PROGRAM prFeedScrewS5
VAR
    SolFeed : fbSingleSolRy;
    ErrorState : BOOL;
    AutoFlow : INT;
    TON1 : TON;
    TON2 : TON;
    TON3 : TON;
    Check1 : fbCheckScrew_Tube;
    Check2 : fbCheckScrew_Tube;
    RTRIG1 : R_TRIG;
END_VAR
VAR_EXTERNAL
    AutoStatus : bool;
    SystemReadyStatus : bool;
    HMIPB_SOL_S5_Feed : BOOL;
    SOL_S5_Feed : BOOL;
    FeedStartFlag : ARRAY[0..1] OF bool;
    HMI_FeedScrewTime : ARRAY[0..1] OF INT;
    RY_S5_Feed : BOOL;
    OutPutFeedRYS5 : BOOL;
    LS_S5_UpDownOut : BOOL;
    SNR_S5_L_Feed : BOOL;
    PB_Reset1 : BOOL;
    PB_Reset2 : BOOL;
    Error_SNR_S5_L_Feed : BOOL;
    SNR_S5_R_Feed : BOOL;
    Error_SNR_S5_R_Feed : BOOL;
    OBJScrewInClip : ARRAY[0..3] OF INT;
    OBJScrewInTube : ARRAY[0..3] OF INT;
    LS_S5_UpDownBack : BOOL;
    SOL_S5_UpDown : BOOL;
    HMIPB_S5Feed : BOOL;
END_VAR
//********************************************************************
//Check
//********************************************************************
Check1(
	inClearSingle:=LS_S5_UpDownOut,
	inFeedSNR:=SNR_S5_L_Feed,
	inBlowSOL:=SOL_S5_Feed,
	inReset:=PB_Reset1 OR PB_Reset2,
	outError=>Error_SNR_S5_L_Feed,
	inoutScrewInClip:=OBJScrewInClip[0],
	inoutScrewInTube:=OBJScrewInTube[0]);
Check2(
	inClearSingle:=LS_S5_UpDownOut,
	inFeedSNR:=SNR_S5_R_Feed,
	inBlowSOL:=SOL_S5_Feed,
	inReset:=PB_Reset1 OR PB_Reset2,
	outError=>Error_SNR_S5_R_Feed,
	inoutScrewInClip:=OBJScrewInClip[1],
	inoutScrewInTube:=OBJScrewInTube[1]);
//********************************************************************
//Manual
//********************************************************************
//Feed screw sol
SolFeed(
	inAutoStatus:=AutoStatus,
	inAutoFlowSet:=AutoFlow=3,
	inAutoFlowReset:=AutoFlow=4,
	inInterLockBack:=TRUE,
	inInterLockOut:=NOT(SOL_S5_UpDown) AND LS_S5_UpDownBack,
	outSol=>	SOL_S5_Feed);
//********************************************************************
//Auto
//********************************************************************
IF LS_S5_UpDownOut AND SOL_S5_UpDown THEN
	FeedStartFlag[0]:=TRUE;
END_IF;
ErrorState:=FALSE;
//power on=0
IF NOT(SystemReadyStatus) OR ErrorState THEN
	AutoFlow:=0;
	FeedStartFlag[0]:=FALSE;
END_IF;
//idle=1
IF AutoFlow=0 AND NOT(NOT(SystemReadyStatus) OR ErrorState) THEN
	AutoFlow:=1;
END_IF;
IF AutoFlow=6 AND NOT(OutPutFeedRYS5) THEN
	AutoFlow:=1;
END_IF;
//Feed RY on=2
RTRIG1(Clk:=HMIPB_SOL_S5_Feed);
IF AutoFlow=1 AND ((FeedStartFlag[0] AND AutoStatus) OR (RTRIG1.Q AND NOT(AutoStatus))) THEN
	AutoFlow:=2;
	OutPutFeedRYS5:=TRUE;
END_IF;
//Feed Sol on=3
TON1(In:=AutoFlow=2 AND RY_S5_Feed, PT:=t#800ms);
//
IF AutoFlow=2 AND TON1.Q THEN
	AutoFlow:=3;
END_IF;
IF AutoFlow=5 AND NOT(TON3.Q) AND FeedStartFlag[0] THEN
	AutoFlow:=3;
END_IF;
//Feed Sol off=4
TON2(In:=AutoFlow=3 AND SOL_S5_Feed, PT:=NanoSecToTime(HMI_FeedScrewTime[0]*100000000));
IF AutoFlow=3 AND ((TON2.Q AND AutoStatus) OR RTRIG1.Q AND NOT(AutoStatus)) THEN
	AutoFlow:=4;
END_IF;
//Feed Finish=5
IF AutoFlow=4 AND NOT(SOL_S5_Feed) THEN
	AutoFlow:=5;
	FeedStartFlag[0]:=FALSE;
END_IF;
//Feed RY off=6
TON3(In:=AutoFlow=5, PT:=t#5s);
IF AutoFlow=5 AND TON3.Q THEN
	AutoFlow:=6;
	OutPutFeedRYS5:=FALSE;
END_IF;
END_PROGRAM

PROGRAM prFeedScrewS6
VAR
    SolFeed : fbSingleSolRy;
    ErrorState : BOOL;
    AutoFlow : INT;
    TON1 : TON;
    TON2 : TON;
    TON3 : TON;
    Check1 : fbCheckScrew_Tube;
    Check2 : fbCheckScrew_Tube;
    RTRIG1 : R_TRIG;
END_VAR
VAR_EXTERNAL
    AutoStatus : bool;
    SystemReadyStatus : bool;
    HMIPB_SOL_S5_Feed : BOOL;
    SOL_S5_Feed : BOOL;
    FeedStartFlag : ARRAY[0..1] OF bool;
    HMI_FeedScrewTime : ARRAY[0..1] OF INT;
    RY_S5_Feed : BOOL;
    OutPutFeedRYS5 : BOOL;
    LS_S5_UpDownOut : BOOL;
    SNR_S5_L_Feed : BOOL;
    PB_Reset1 : BOOL;
    PB_Reset2 : BOOL;
    Error_SNR_S5_L_Feed : BOOL;
    SNR_S5_R_Feed : BOOL;
    Error_SNR_S5_R_Feed : BOOL;
    LS_S6_UpDownOut : BOOL;
    SNR_S6_L_Feed : BOOL;
    SOL_S6_Feed : BOOL;
    Error_SNR_S6_L_Feed : BOOL;
    SNR_S6_R_Feed : BOOL;
    Error_SNR_S6_R_Feed : BOOL;
    HMIPB_SOL_S6_Feed : BOOL;
    RY_S6_Feed : BOOL;
    OutPutFeedRYS6 : BOOL;
    OBJScrewInClip : ARRAY[0..3] OF INT;
    OBJScrewInTube : ARRAY[0..3] OF INT;
    LS_S6_UpDownBack : BOOL;
    SOL_S2_Fix : BOOL;
    SOL_S6_UpDown : BOOL;
END_VAR
//********************************************************************
//Check
//********************************************************************
Check1(
	inClearSingle:=LS_S6_UpDownOut,
	inFeedSNR:=SNR_S6_L_Feed,
	inBlowSOL:=SOL_S6_Feed,
	inReset:=PB_Reset1 OR PB_Reset2,
	outError=>Error_SNR_S6_L_Feed,
	inoutScrewInClip:=OBJScrewInClip[2],
	inoutScrewInTube:=OBJScrewInTube[2]);
Check2(
	inClearSingle:=LS_S6_UpDownOut,
	inFeedSNR:=SNR_S6_R_Feed,
	inBlowSOL:=SOL_S6_Feed,
	inReset:=PB_Reset1 OR PB_Reset2,
	outError=>Error_SNR_S6_R_Feed,
	inoutScrewInClip:=OBJScrewInClip[3],
	inoutScrewInTube:=OBJScrewInTube[3]);
//********************************************************************
//Manual
//********************************************************************
//Feed screw sol
SolFeed(
	inAutoStatus:=AutoStatus,
	inAutoFlowSet:=AutoFlow=3,
	inAutoFlowReset:=AutoFlow=4,
	inInterLockBack:=TRUE,
	inInterLockOut:=NOT(SOL_S6_UpDown) AND LS_S6_UpDownBack,
	outSol=>	SOL_S6_Feed);
//********************************************************************
//Auto
//********************************************************************
IF LS_S6_UpDownOut AND SOL_S6_UpDown THEN
	FeedStartFlag[1]:=TRUE;
END_IF;
ErrorState:=FALSE;
//power on=0
IF NOT(SystemReadyStatus) OR ErrorState THEN
	AutoFlow:=0;
	FeedStartFlag[1]:=FALSE;
END_IF;
//idle=1
IF AutoFlow=0 AND NOT(NOT(SystemReadyStatus) OR ErrorState) THEN
	AutoFlow:=1;
END_IF;
IF AutoFlow=6 AND NOT(OutPutFeedRYS6) THEN
	AutoFlow:=1;
END_IF;
//Feed RY on=2
RTRIG1(Clk:=HMIPB_SOL_S6_Feed);
IF AutoFlow=1 AND ((FeedStartFlag[1] AND AutoStatus) OR (RTRIG1.Q AND NOT(AutoStatus))) THEN
	AutoFlow:=2;
	OutPutFeedRYS6:=TRUE;
END_IF;
//Feed Sol on=3
TON1(In:=AutoFlow=2 AND RY_S6_Feed, PT:=t#800ms);
//
IF AutoFlow=2 AND TON1.Q THEN
	AutoFlow:=3;
END_IF;
IF AutoFlow=5 AND NOT(TON3.Q) AND FeedStartFlag[1] THEN
	AutoFlow:=3;
END_IF;
//Feed Sol off=4
TON2(In:=AutoFlow=3 AND SOL_S6_Feed, PT:=NanoSecToTime(HMI_FeedScrewTime[1]*100000000));
IF AutoFlow=3 AND ((TON2.Q AND AutoStatus) OR RTRIG1.Q AND NOT(AutoStatus)) THEN
	AutoFlow:=4;
END_IF;
//Feed Finish=5
IF AutoFlow=4 AND NOT(SOL_S6_Feed) THEN
	AutoFlow:=5;
	FeedStartFlag[1]:=FALSE;
END_IF;
//Feed RY off=6
TON3(In:=AutoFlow=5, PT:=t#5s);
IF AutoFlow=5 AND TON3.Q THEN
	AutoFlow:=6;
	OutPutFeedRYS6:=FALSE;
END_IF;
END_PROGRAM

PROGRAM prCommProgram
VAR
    statusFlash1s : BOOL;
    bClock : BOOL;
    TON1 : TON;
    TON2 : TON;
    R_TRIG1 : R_TRIG;
END_VAR
VAR_EXTERNAL
    Flash1s : BOOL;
    HMIPB_ResetCount : BOOL;
    HMI_AllCount : UDINT;
END_VAR
//bClock:=Get1sClk();
IF HMIPB_ResetCount THEN
	HMI_AllCount:=0;
END_IF;
//flsash 1s
TON1(In:=NOT(statusFlash1s), PT:=t#1s);
TON2(In:=(statusFlash1s), PT:=t#1s);
IF TON1.Q THEN
	bClock:=TRUE;
END_IF;
IF TON2.Q THEN
	bClock:=FALSE;
END_IF;
Flash1s:=bClock;
statusFlash1s:=Flash1s;
END_PROGRAM

PROGRAM prBZAndLight
VAR_EXTERNAL
    Flash1s : BOOL;
    GL : BOOL;
    YL : BOOL;
    SystemReadyStatus : bool;
    ErrorStatus_MachineNonStop : bool;
    ErrorStatus_MachineStop : bool;
    RL : BOOL;
    BZ : BOOL;
    MachineRunStatus : bool;
END_VAR
(*BZ*)	
IF (ErrorStatus_MachineStop OR ErrorStatus_MachineNonStop) THEN
	BZ:=Flash1s;
	ELSE
	BZ:=FALSE;
END_IF;
//(*紅燈長亮:異常*)
IF SystemReadyStatus AND (ErrorStatus_MachineStop) THEN
	RL:=TRUE;
	ELSE
	RL:=FALSE;
END_IF;
(*綠燈閃爍:運轉,長亮:待機*)
IF SystemReadyStatus AND NOT(ErrorStatus_MachineNonStop) AND NOT(ErrorStatus_MachineStop)  THEN
	IF MachineRunStatus THEN
		GL:=Flash1s;
	ELSE
		GL:=TRUE;
	END_IF;
	ELSE
	GL:=FALSE;
END_IF;
(*黃燈閃爍:振動筒缺料*)
IF SystemReadyStatus AND ErrorStatus_MachineNonStop AND NOT(ErrorStatus_MachineStop) THEN
	YL:=Flash1s;
	ELSE
	YL:=FALSE;
END_IF;
END_PROGRAM

PROGRAM prCycleTime
VAR
    TON1 : TON;
    tCycleTime : TIME;
    RTRIG1 : R_TRIG;
    cycle : LINT;
    FTRIG1 : F_TRIG;
END_VAR
VAR_EXTERNAL
    HMI_CycleTime : LINT;
    MachineRunStatus : bool;
    SNR_Index : BOOL;
END_VAR
IF FTRIG1.Q THEN
	HMI_CycleTime:=cycle;
END_IF;
TON1(In:=MachineRunStatus AND SNR_Index, PT:=t#1m,ET=>tCycleTime);
IF MachineRunStatus AND SNR_Index THEN
	cycle:=TimeToNanoSec(tCycleTime)/10000000;
END_IF;
FTRIG1(Clk:=SNR_Index);
END_PROGRAM

FUNCTION fIndexDataChange : BOOL
VAR_EXTERNAL
    IndexData8 : StationRecord;
    IndexData7 : StationRecord;
    IndexData6 : StationRecord;
    IndexData5 : StationRecord;
    IndexData4 : StationRecord;
    IndexData3 : StationRecord;
    IndexData2 : StationRecord;
    IndexData1 : StationRecord;
    IndexData0 : StationRecord;
END_VAR
IndexData8:=IndexData7;
IndexData7:=IndexData6;
IndexData6:=IndexData5;
IndexData5:=IndexData4;
IndexData4:=IndexData3;
IndexData3:=IndexData2;
IndexData2:=IndexData1;
IndexData1:=IndexData0;
END_FUNCTION

FUNCTION_BLOCK fbBowlFeeder
VAR
    AutoFlow : INT;
    TON_Auto1 : TON;
    TON_Auto2 : TON;
    TON_Auto3 : TON;
    tItemNotExistDelayTime : TIME;
    tItemExistTime : TIME;
    tItemNotExistErrorTime : TIME;
END_VAR
VAR_INPUT
    bFullSNR : BOOL;
    iItemNotExistDelayTime : LINT;
    iItemExistTime : LINT;
    iItemNotExistErrorTime : LINT;
END_VAR
VAR_OUTPUT
    bFullRY : BOOL;
    bFullSNRError : BOOL;
END_VAR
VAR_EXTERNAL
    SystemReadyStatus : BOOL;
END_VAR
(******************************************************************
程式:振動筒程序
作者:蔡相偉
版本資訊:v1.0		2016/4/16
******************************************************************)
//時間轉換
tItemNotExistDelayTime:=NanoSecToTime(In:=iItemNotExistDelayTime*100000000);
tItemExistTime:=NanoSecToTime(In:=iItemExistTime*100000000);
tItemNotExistErrorTime:=NanoSecToTime(In:=iItemNotExistErrorTime*100000000);
(*流程*)
(*PowerOn=0*)
IF NOT(SystemReadyStatus) THEN
	AutoFlow:=0;
END_IF;

(*Idle=1*)
IF AutoFlow=0 AND SystemReadyStatus THEN
	AutoFlow:=1;
END_IF;

IF AutoFlow=3 THEN
	AutoFlow:=1;
END_IF;

(*振動筒起振=2*)
TON_Auto1(IN:=AutoFlow=1 AND NOT(bFullSNR) , PT:=tItemNotExistDelayTime);
IF AutoFlow=1 AND TON_Auto1.Q THEN
	AutoFlow:=2;
END_IF;

(*振動筒停振=3*)
TON_Auto2(IN:=AutoFlow=2 AND bFullSNR , PT:=tItemExistTime);
TON_Auto3(IN:=NOT(bFullSNR) AND bFullRY, PT:=tItemNotExistErrorTime);
IF AutoFlow=2 AND TON_Auto2.Q THEN
	AutoFlow:=3;
END_IF;
(******************************************************************)
(*輸出*)
(*振動筒繼電器*)
IF AutoFlow=2 THEN
	bFullRY:=TRUE;
	ELSE
	bFullRY:=FALSE;
END_IF;
(*振動筒滿料異常*)
IF AutoFlow=2 AND (TON_Auto3.Q) THEN
	bFullSNRError:=TRUE;
	ELSE
	bFullSNRError:=FALSE;
END_IF;
END_FUNCTION_BLOCK

FUNCTION_BLOCK fbSingleSolRy
VAR
    solStatus : BOOL;
    R_TRIG1 : R_TRIG;
END_VAR
VAR_INPUT
    inPushButton : BOOL;
    inAutoStatus : BOOL;
    inAutoFlowSet : BOOL;
    inAutoFlowReset : BOOL;
    inInterLockBack : BOOL;
    inInterLockOut : BOOL;
END_VAR
VAR_OUTPUT
    outSol : BOOL;
END_VAR
(*電磁閥*)
R_TRIG1(Clk:=inPushButton AND NOT(inAutoStatus));
(*SET*)
IF ((R_TRIG1.Q AND NOT(solStatus)) OR inAutoFlowSet) AND inInterLockOut THEN
	outSol:=TRUE;
END_IF;
(*RESET*)
IF ((R_TRIG1.Q AND (solStatus)) OR inAutoFlowReset) AND inInterLockBack THEN
	outSol:=FALSE;
END_IF;
(*STATUS*)
solStatus:=outSol;
END_FUNCTION_BLOCK

FUNCTION_BLOCK fbErrorSOL_S
VAR
    TON_1 : TON;
    TON_2 : TON;
END_VAR
VAR_INPUT
    bAutoStatus : BOOL;
    bResetPB : BOOL;
    bSOL : BOOL;
    bBackLS : BOOL;
    bOutLS : BOOL;
END_VAR
VAR_OUTPUT
    bErrorStatus_Back : BOOL;
    bErrorStatus_Out : BOOL;
END_VAR
IF bAutoStatus AND NOT(bResetPB) THEN
	(*歸磁簧開關*)
	TON_1(IN:=(NOT(bSOL) AND NOT(bBackLS)) OR ((bSOL) AND bBackLS), PT:=t#2s);
	IF TON_1.Q THEN
		bErrorStatus_Back:=TRUE;
	END_IF;
	(*出磁簧開關*)
	TON_2(IN:=(NOT(bSOL) AND (bOutLS)) OR ((bSOL) AND NOT(bOutLS)), PT:=t#2s);
	IF TON_2.Q THEN
		bErrorStatus_Out:=TRUE;
	END_IF;
END_IF;
IF bResetPB THEN
	bErrorStatus_Back:=FALSE;
	bErrorStatus_Out:=FALSE;
END_IF;
END_FUNCTION_BLOCK

FUNCTION_BLOCK fbErrorSOL_D
VAR
    TON_1 : TON;
    TON_2 : TON;
END_VAR
VAR_INPUT
    bAutoStatus : BOOL;
    bResetPB : BOOL;
    bBackSOL : BOOL;
    bOutSOL : BOOL;
    bBackLS : BOOL;
    bOutLS : BOOL;
END_VAR
VAR_OUTPUT
    bErrorStatus_Back : BOOL;
    bErrorStatus_Out : BOOL;
END_VAR
IF bAutoStatus AND NOT(bResetPB) THEN
	(*歸磁簧開關*)
	TON_1(IN:=bBackSOL AND NOT(bBackLS), PT:=t#4s);
	IF TON_1.Q THEN
		bErrorStatus_Back:=TRUE;
	END_IF;
	(*出磁簧開關*)
	TON_2(IN:=bOutSOL AND NOT(bOutLS), PT:=t#4s);
	IF TON_2.Q THEN
		bErrorStatus_Out:=TRUE;
	END_IF;
END_IF;
IF bResetPB THEN
	bErrorStatus_Back:=FALSE;
	bErrorStatus_Out:=FALSE;
END_IF;
END_FUNCTION_BLOCK

FUNCTION_BLOCK fbCheckScrew_Clamp
VAR
    R_TRIG1 : R_TRIG;
    R_TRIG2 : R_TRIG;
    F_TRIG1 : F_TRIG;
END_VAR
VAR_INPUT
    inClearSingle : BOOL;
    inFeedSNR : BOOL;
    inBlowSOL : BOOL;
    inReset : BOOL;
END_VAR
VAR_OUTPUT
    outError : BOOL;
END_VAR
VAR_IN_OUT
    inoutScrewInClip : INT;
END_VAR
R_TRIG1(CLK:= inClearSingle);
R_TRIG2(CLK:= inFeedSNR);
F_TRIG1(Clk:=inBlowSOL);

IF R_TRIG2.Q THEN
	inoutScrewInClip:=inoutScrewInClip+1;
END_IF;

IF R_TRIG1.Q THEN
	inoutScrewInClip:=0;
END_IF;

IF F_TRIG1.Q AND inoutScrewInClip<=0 THEN
	outError:=TRUE;
END_IF;
IF inReset THEN
	outError:=FALSE;
END_IF;
END_FUNCTION_BLOCK

FUNCTION_BLOCK fbDoubleSolRy
VAR_INPUT
    inPushBackButton : BOOL;
    inPushOutButton : BOOL;
    inAutoStatus : BOOL;
    inAutoFlowSet : BOOL;
    inAutoFlowReset : BOOL;
    inInterLockBack : BOOL;
    inInterLockOut : BOOL;
    inBackSensor : BOOL;
    inOutSensor : BOOL;
END_VAR
VAR_OUTPUT
    outBackSol : BOOL;
    outOutSol : BOOL;
END_VAR
(*Out電磁閥*)
IF (inPushOutButton OR inAutoFlowSet) AND inInterLockOut THEN
	outOutSol:=TRUE;
	outBackSol:=FALSE;
END_IF;
IF inOutSensor THEN
	outOutSol:=FALSE;
END_IF;
(*Back電磁閥*)
IF (inPushBackButton OR inAutoFlowReset) AND inInterLockBack THEN
	outOutSol:=FALSE;
	outBackSol:=TRUE;
END_IF;
IF inBackSensor THEN
	outBackSol:=FALSE;
END_IF;
END_FUNCTION_BLOCK

FUNCTION_BLOCK fbCheckScrew_Tube
VAR
    R_TRIG1 : R_TRIG;
    R_TRIG2 : R_TRIG;
    R_TRIG3 : R_TRIG;
    F_TRIG1 : F_TRIG;
END_VAR
VAR_INPUT
    inClearSingle : BOOL;
    inFeedSNR : BOOL;
    inBlowSOL : BOOL;
    inReset : BOOL;
END_VAR
VAR_OUTPUT
    outError : BOOL;
END_VAR
VAR_IN_OUT
    inoutScrewInClip : INT;
    inoutScrewInTube : INT;
END_VAR
R_TRIG1(CLK:= inClearSingle);
R_TRIG2(CLK:= inFeedSNR);
R_TRIG3(CLK:= inBlowSOL);
F_TRIG1(Clk:=inBlowSOL);

IF R_TRIG2.Q THEN
	inoutScrewInTube:=inoutScrewInTube+1;
END_IF;

IF R_TRIG1.Q THEN
	inoutScrewInClip:=0;
END_IF;

IF R_TRIG3.Q THEN
	inoutScrewInClip:=inoutScrewInTube;
	inoutScrewInTube:=0;
END_IF;

IF F_TRIG1.Q AND inoutScrewInClip<=0 THEN
	outError:=TRUE;
END_IF;
IF inReset THEN
	outError:=FALSE;
END_IF;
END_FUNCTION_BLOCK

FUNCTION_BLOCK fbScrewFlow
VAR
    AutoFlow : INT;
    TONNG : TON;
    TON7 : TON;
    TON20 : TON;
    TON30 : TON;
    oldTorque : LREAL;
    torquecount : INT;
    sensorONFlag : BOOL;
END_VAR
VAR_INPUT
    inStartFlag : BOOL;  (* 起動 *)
    inCheckSensor : BOOL;  (* 檢查近接開關 *)
    inStopFlag : BOOL;  (* standstill *)
    inBackoutBusy : BOOL;  (* busy *)
    inCMDTorque : LREAL;  (* 退扭力 *)
    inCMDAddress : LREAL;  (* 下鎖限制角度 *)
    inNoScrewSetAngle : LREAL;  (* 無螺絲檢查角度 *)
    inFindTime : LINT;  (* 反轉時間 *)
    inTorqueValue : LREAL;  (* 扭力顯示 *)
    inAddressValue : LREAL;  (* 角度顯示 *)
END_VAR
VAR_OUTPUT
    outFW : BOOL;  (* 正轉PB *)
    outRW : BOOL;  (* 反轉PB *)
    outBackout : BOOL;  (* Backout Start *)
    outFlowNo : INT;  (* 當前流程碼 *)
    outResetAddress : BOOL;  (* HOME PB *)
END_VAR
VAR_IN_OUT
    inoutTorque : LREAL;  (* 下鎖扭力設定值 *)
END_VAR
VAR_EXTERNAL
    SystemReadyStatus : bool;
END_VAR
VAR_EXTERNAL CONSTANT
    MC_AxisLSt5 : _sAXIS_REF;
END_VAR
//power on
IF NOT(SystemReadyStatus) THEN
	AutoFlow:=0;
END_IF;
//idle
IF AutoFlow=0 AND SystemReadyStatus THEN
	AutoFlow:=1;
END_IF;
IF AutoFlow=8 AND NOT(outRW) AND NOT(inStartFlag) AND oldTorque=inoutTorque THEN
	AutoFlow:=1;
END_IF;
IF AutoFlow=9999 AND NOT(outFW) AND NOT(inStartFlag) AND oldTorque=inoutTorque  THEN
	AutoFlow:=1;
END_IF;
//反轉=30
IF AutoFlow=1 AND inStartFlag THEN
	torquecount:=0;
	oldTorque:=inoutTorque;
	outResetAddress:=TRUE;
	sensorONFlag:=FALSE;
	outRW:=TRUE;
	AutoFlow:=30;
END_IF;
//停止=31
TON30(In:=AutoFlow=30 AND outRW, PT:=NanoSecToTime(In:=inFindTime*100000000));
IF AutoFlow=30 AND TON30.Q THEN
    outRW:=FALSE;
	AutoFlow:=31;
END_IF;
//set 0 on=20
IF AutoFlow=31 AND NOT(outRW) AND inStopFlag THEN
	AutoFlow:=20;
END_IF;
//set0 off=21
TON20(In:=AutoFlow=20 AND outResetAddress,PT:=t#300ms);
IF AutoFlow=20 AND TON20.Q THEN
	outResetAddress:=FALSE;
	AutoFlow:=21;
END_IF;
//起動=2
IF AutoFlow=21 AND NOT(outResetAddress) THEN
	outFW:=TRUE;
	AutoFlow:=2;
END_IF;
//snesor到達=3
IF AutoFlow=2 AND inCheckSensor AND NOT(TONNG.Q) THEN
	AutoFlow:=3;
END_IF;
//snesor未到達=9999
TONNG(In:=AutoFlow>=2 AND AutoFlow<9000,PT:=t#6s);
IF AutoFlow>=2 AND TONNG.Q THEN
	outFW:=FALSE;
	outRW:=FALSE;
	inoutTorque:=oldTorque;
	AutoFlow:=9999;
END_IF;
IF AutoFlow=2 AND (inAddressValue>=inCMDAddress) AND oldTorque=inoutTorque THEN
	outFW:=FALSE;
	outRW:=FALSE;
	inoutTorque:=oldTorque;
	AutoFlow:=9999;
END_IF;
IF inCheckSensor THEN
	sensorONFlag:=TRUE;
END_IF;

//停止=4
IF AutoFlow=3 AND inCheckSensor THEN
	outFW:=FALSE;
	AutoFlow:=4;
END_IF;
//設定=5
IF AutoFlow=4 AND NOT(outFW) THEN
	AutoFlow:=5;
END_IF;
//反轉=6
IF AutoFlow=5 AND inStopFlag THEN
	outBackout:=TRUE;
	AutoFlow:=6;
END_IF;
//反轉中=7
IF AutoFlow=6 AND inBackoutBusy THEN
	outBackout:=FALSE;
	AutoFlow:=7;
END_IF;
//停止=8
IF AutoFlow=7 AND NOT(inBackoutBusy) AND NOT(outRW) THEN
	AutoFlow:=8;
END_IF;
outFlowNo:=AutoFlow;
END_FUNCTION_BLOCK